TYPE E_FILE_CtrlState :
(
	E_CX_FILEIDLE,
	E_CX_FILEOPEN,
	E_CX_FILESEEK,
	E_CX_FILEREAD,
	E_CX_FILEWRITE,
	E_CX_FILECLOSE,
	E_CX_FILEDONE
);
END_TYPE

(* stored: Version 1.1.0.1, ProductVersion 3.1.4024.15
   DUT E_FILE_CtrlState: Id {99960360-056d-4d9c-81cc-e92f2896876d} *)
